Yaskawa INFORM job: OK_R2_O50&56(110_90,0)AWOK.JBI

/JOB
//NAME OK_R2_O50&56(110_90,0)AWOK
///FOLDERNAME X4
//POS
///NPOS 283,283,283,16,0,0
///TOOL 0
///POSTYPE PULSE
///PULSE
C00000=-174960,-106597,-120103,-3797,95090,7084
C00001=-145942,12948,-48978,-9200,114636,15117
C00002=-148771,199,-24149,-7829,92768,15748
C00003=-149791,3169,-18240,-7666,90580,15544
C00004=-150189,4428,-15804,-7606,89698,15465
C00005=-150189,4377,-14625,-7604,88953,15510
C00006=-150189,4428,-15804,-7606,89698,15465
C00007=-147129,1088,-19588,-8038,90597,16430
C00008=-146286,3274,-14174,-8147,88492,16849
C00009=-147032,3892,-13646,-8045,88411,16604
C00010=-146286,3274,-14174,-8147,88492,16849
C00011=-145329,9981,-8228,-8277,88377,17179
C00012=-145001,12478,-5992,-8324,88322,17293
C00013=-145329,9981,-8228,-8277,88377,17179
C00014=-145885,10408,-7967,-8202,88379,16992
C00015=-146004,9179,-11468,-8189,89874,16853
C00016=-148771,199,-24149,-7829,92768,15748
C00017=-146250,12959,-11588,-41426,106240,56782
C00018=-148467,10115,-11951,-41164,104276,56589
C00019=-154824,5653,-21154,-31285,103371,55685
C00020=-154824,5441,-20026,-31169,102684,55881
C00021=-149371,9046,-12025,-41064,103475,56508
C00022=-146311,6118,-11326,-40674,103401,57916
C00023=-147454,7095,-10477,-40693,102859,57619
C00024=-146311,6118,-11326,-40674,103401,57916
C00025=-146151,4867,-13193,-40766,103863,57802
C00026=-146384,3242,-14587,-40774,103772,57733
C00027=-146151,4867,-13193,-40766,103863,57802
C00028=-145246,5991,-13096,-40848,104676,57882
C00029=-143030,9240,-15326,-41491,108018,57509
C00030=-124603,-47737,-34158,19131,104982,-62056
C00031=-121442,-51513,-32422,19687,101389,-61480
C00032=-118855,-51471,-32397,20347,100766,-60636
C00033=-118855,-50574,-30118,20274,99880,-60787
C00034=-118855,-51471,-32397,20347,100766,-60636
C00035=-121442,-51513,-32422,19687,101389,-61480
C00036=-121797,-50324,-29168,19487,100158,-61813
C00037=-120620,-50331,-29171,19792,99877,-61431
C00038=-121797,-50324,-29168,19487,100158,-61813
C00039=-121442,-51513,-32422,19687,101389,-61480
C00040=-121603,-51176,-29855,19536,100099,-61752
C00041=-121615,-53238,-31000,19508,99766,-61811
C00042=-121603,-51176,-29855,19536,100099,-61752
C00043=-122128,-47866,-34232,19785,104374,-61232
C00044=-84141,-29178,-36607,14646,114104,-67707
C00045=-82791,-33286,-36430,14724,111710,-67503
C00046=-82229,-34853,-36282,14765,110740,-67415
C00047=-82178,-34515,-34630,14688,109914,-67503
C00048=-82229,-34853,-36282,14765,110740,-67415
C00049=-79147,-30434,-31070,15425,109262,-66446
C00050=-78452,-32631,-32544,15567,108914,-66232
C00051=-79147,-30434,-31070,15425,109262,-66446
C00052=-79730,-28966,-31252,15378,110209,-66539
C00053=-81132,-25108,-31519,15285,112547,-66756
C00054=-131359,-62866,-74976,11014,90207,-78232
C00055=-138536,21396,-13882,13391,108121,-66751
C00056=-115516,26685,-4177,3986,97138,-31002
C00057=-94522,36317,14190,8701,90062,-23707
C00058=-87387,60420,45294,7806,89491,-21265
C00059=-87081,59268,47156,7800,87741,-21270
C00060=-87136,59191,47136,7801,87720,-21290
C00061=-87136,59626,48812,7802,86921,-21339
C00062=-87136,58571,44510,7803,89008,-21209
C00063=-94386,48885,37947,21340,84274,-24043
C00064=-93739,49715,38851,21295,83986,-23861
C00065=-94392,49010,38218,21343,84180,-24062
C00066=-94392,48026,33496,21296,86424,-23665
C00067=-99028,41403,18475,21708,93080,-24149
C00068=-102045,-22247,-40217,22084,97043,-24505
C00069=-74840,-13391,-38223,2617,97503,-17820
C00070=-66507,5010,-12577,-6934,97902,-16018
C00071=-66195,5774,-8292,-6895,95700,-15788
C00072=-66101,6043,-7102,-6886,95120,-15724
C00073=-66101,6129,-6115,-6879,94563,-15693
C00074=-66101,5877,-9999,-6916,96808,-15817
C00075=-80836,-17286,-23478,14204,80508,-20001
C00076=-80064,-16344,-22775,14064,80424,-19740
C00077=-80850,-17465,-25526,14169,81645,-19874
C00078=-68799,5840,-15749,-112,106098,-15895
C00079=-55050,-26211,-40797,896,104976,-11120
C00080=-53240,-26394,-33808,1003,100562,-10527
C00081=-53174,-26119,-32540,1008,99922,-10509
C00082=-53174,-26003,-31510,1007,99347,-10512
C00083=-53450,-26813,-34326,989,100667,-10598
C00084=-66076,-50527,-45741,15470,82986,-15464
C00085=-65365,-49438,-45112,15396,83017,-15209
C00086=-66444,-51488,-48366,15481,84138,-15447
C00087=-76298,-64666,-67677,16335,90985,-18012
C00088=-121005,-146046,-93198,13283,20086,50099
C00089=-121076,-175637,-121627,12100,22333,50657
C00090=-121076,-175637,-121627,12100,22333,50657
C00091=-119842,-145846,-119955,-19490,98596,-44269
C00092=-120072,-86643,-91493,-20899,110694,-78316
C00093=-121200,-92303,-90459,-20559,107088,-78084
C00094=-138616,-107413,-91097,-21806,95703,-82500
C00095=-138616,-107085,-90210,-21788,95350,-82435
C00096=-138616,-107413,-91097,-21806,95703,-82500
C00097=-139134,-110877,-92284,-21800,94587,-82488
C00098=-138616,-107413,-91097,-21806,95703,-82500
C00099=-138504,-107678,-93902,-21887,97214,-82736
C00100=-111033,-68243,-79959,-15660,119373,-68405
C00101=-111039,-68171,-79817,-15653,119324,-68399
C00102=-111039,-68347,-78629,-15518,118531,-68280
C00103=-111039,-68171,-79817,-15653,119324,-68399
C00104=-110811,-71611,-81502,-15474,118663,-68211
C00105=-111039,-68171,-79817,-15653,119324,-68399
C00106=-117681,-73428,-89845,-994,113898,-68956
C00107=-117328,-75555,-88746,-937,112132,-68814
C00108=-117314,-76363,-88422,-931,111517,-68804
C00109=-117314,-76477,-87912,-929,111141,-68802
C00110=-117314,-76038,-89659,-939,112445,-68812
C00111=-117225,-80228,-90181,-914,110615,-68766
C00112=-117357,-73687,-89896,-955,113798,-68838
C00113=-117304,-75426,-92745,-956,114658,-68828
C00114=-117163,-75550,-92733,-938,114587,-68776
C00115=-117163,-75975,-91679,-932,113721,-68770
C00116=-117163,-75740,-92281,-935,114212,-68773
C00117=-117065,-80067,-94252,-916,113200,-68731
C00118=-117163,-75740,-92281,-935,114212,-68773
C00119=-126928,-93462,-104099,21125,97375,-56056
C00120=-123436,-95743,-101732,20630,94052,-55403
C00121=-119720,-93386,-98939,20195,92672,-54328
C00122=-119720,-93542,-97538,20172,91785,-54475
C00123=-119720,-93459,-98367,20185,92306,-54389
C00124=-117930,-93370,-98332,19971,91899,-53827
C00125=-119720,-93459,-98367,20185,92306,-54389
C00126=-119671,-100746,-101187,20141,90406,-54690
C00127=-119720,-93459,-98367,20185,92306,-54389
C00128=-121215,-96042,-102269,20389,93677,-54685
C00129=-124737,-93931,-104706,20902,96960,-55358
C00130=-120615,-97600,-94225,24394,68229,-41312
C00131=-121614,-94302,-98325,24715,72989,-35072
C00132=-121413,-94319,-98186,24655,72844,-35027
C00133=-121413,-94400,-96939,24754,72105,-35186
C00134=-121413,-94319,-98186,24655,72844,-35027
C00135=-119573,-94306,-98179,23998,72315,-34443
C00136=-121413,-94319,-98186,24655,72844,-35027
C00137=-131582,-92162,-101045,27739,78553,-37534
C00138=-149979,-79190,-101251,32758,90741,-41130
C00139=-131734,108486,68329,27886,77598,-37823
C00140=-131746,115175,77213,28093,75801,-38268
C00141=-128705,103754,56939,17355,80936,-37498
C00142=-126391,103513,58781,16629,79272,-36943
C00143=-126391,103204,59430,16657,78740,-37018
C00144=-126391,103325,59164,16645,78953,-36987
C00145=-131461,101888,64135,32515,75623,-37675
C00146=-130460,102804,65331,32242,75027,-37451
C00147=-132956,104856,68008,33106,75465,-38321
C00148=-123747,88520,39161,14959,81804,-36039
C00149=-123722,90598,43933,15013,79993,-36251
C00150=-123722,90479,44118,15020,79823,-36272
C00151=-123708,91557,46446,15056,78971,-36374
C00152=-123735,88704,42579,15029,79860,-36272
C00153=-122122,90222,44481,14459,79203,-35813
C00154=-121873,91643,46282,14382,78796,-35780
C00155=-122407,90627,44476,14554,79458,-35880
C00156=-127598,110669,63569,17480,87727,-36370
C00157=-127458,127775,88290,17571,81562,-37206
C00158=-126717,107110,60862,17217,87970,-36047
C00159=-121872,67125,15966,8400,79107,-26604
C00160=-119947,67886,17918,7577,78131,-26061
C00161=-121414,74104,25465,6223,76455,-25162
C00162=-123564,69808,18958,7132,78404,-25740
C00163=-121169,67878,17908,8113,78241,-26441
C00164=-119911,67888,17920,7562,78127,-26050
C00165=-118039,62377,14643,6757,77165,-25512
C00166=-118781,60315,11658,7068,77995,-25701
C00167=-123961,59152,819,9198,84481,-26863
C00168=-132618,-110497,-108947,28734,74981,-37704
C00169=-124566,-101520,-102656,26093,73034,-35072
C00170=-120616,-96463,-99082,24682,72208,-33752
C00171=-122368,-97019,-90544,25347,66960,-42290
C00172=-120612,-98338,-92224,24658,66756,-41637
C00173=-120867,-94497,-89822,24667,67282,-41619
C00174=-120867,-94581,-89855,24671,67261,-41624
C00175=-125926,-44970,-69160,31039,100350,-58621
C00176=-113068,-21348,-59770,17386,114865,-66123
C00177=-116612,-26527,-62656,17238,114697,-67420
C00178=-116612,-22676,-66743,18014,118989,-66712
C00179=-96791,-67830,-88966,12124,96584,-58954
C00180=-96132,-69249,-87303,11968,94777,-58911
C00181=-126837,-94677,-94277,15990,96379,-69031
C00182=-126113,-98665,-96629,15951,95659,-68871
C00183=-122876,-86143,-90735,14433,101585,-73815
C00184=-123356,-88352,-92131,14143,100582,-73012
C00185=-123771,-89216,-91995,14110,100142,-73211
C00186=-120613,-99078,-98492,7508,100072,-69302
C00187=-121484,-95136,-96163,7500,100739,-69561
C00188=-172923,-99461,-89995,9994,101945,-90389
C00189=-177663,-102072,-90824,8800,99779,-89697
C00190=-154720,-73630,-87216,6031,109011,-80641
C00191=-161015,-76454,-86164,5490,107360,-82931
C00192=-120149,-70168,-111353,-20212,74375,-72326
C00193=-120057,-133921,-120473,-34069,36215,-62022
C00194=-120146,-106815,-117651,-27009,46787,-66237
C00195=-120793,-117832,-87628,-5856,54262,2374
C00196=-128370,-47930,-37102,-5352,91873,78331
C00197=-120655,-51136,-30966,-4745,86952,81146
C00198=-120656,-51126,-30961,-4745,86954,81145
C00199=-121240,-72948,-42427,-4950,70443,81585
C00200=-120654,-52833,-32998,-4744,87329,81132
C00201=-120662,-49043,-29779,-4745,87295,81131
C00202=-130317,-72190,-42085,-4090,70120,78412
C00203=-120656,-51164,-30982,-4745,86947,81145
C00204=-120655,-51174,-30987,-4745,86946,81146
C00205=-120663,-45936,-34749,-4755,91934,80956
C00206=-120658,-53922,-38518,13016,106165,-78731
C00207=-120658,-51068,-30928,12795,103038,-79070
C00208=-120848,-68568,-43477,12343,92645,-80201
C00209=-120664,-48985,-29748,12815,103375,-79036
C00210=-120728,-51718,-32595,12818,103725,-79022
C00211=-121033,-67565,-42727,12320,93337,-80192
C00212=-120658,-51052,-30919,12796,103041,-79070
C00213=-120658,-51066,-30927,12796,103039,-79070
C00214=-93952,-51121,-30967,10241,104523,67822
C00215=-93953,-51118,-30965,10240,104524,67822
C00216=-94232,-51834,-31148,10139,104305,67705
C00217=-94418,-49164,-29853,10109,104897,67688
C00218=-92862,-50813,-31445,10614,104829,68238
C00219=-94060,-51719,-30968,10193,104235,67762
C00220=-94696,-51466,-31161,9999,104558,67560
C00221=-98759,-53921,-36367,8775,106946,66293
C00222=-98759,-54646,-38349,8822,107784,66355
C00223=-121493,-81341,-55216,13751,94719,-44592
C00224=-114524,-75581,-43376,14967,89304,-42820
C00225=-114061,-74120,-39769,15046,87799,-42845
C00226=-113295,-83137,-43502,15198,85402,-42879
C00227=-116252,-82247,-47187,14646,88567,-43499
C00228=-99157,-63031,-38155,9295,97620,-77423
C00229=-98614,-64282,-34857,9364,94917,-77440
C00230=-110866,-75942,-40129,15794,87673,-68088
C00231=-113165,-74166,-45037,15395,91900,-68341
C00232=-115008,-93546,-53723,13756,68589,-42068
C00233=-109675,-90309,-49025,11903,66648,-40175
C00234=-110872,-80814,-45342,11782,69375,-40325
C00235=-112821,-83961,-50903,11792,71421,-40812
C00236=-114232,-64224,-42018,11630,76204,-40845
C00237=-112624,-62061,-36751,11627,73886,-40501
C00238=-113161,-53891,-32402,11587,75454,-40540
C00239=-113879,-55267,-35641,11577,76817,-40664
C00240=-113966,-53043,-33005,11293,67484,-41540
C00241=-113291,-51178,-29635,11252,66296,-41408
C00242=-111200,-67941,-30076,11904,38840,-43371
C00243=-111272,-77572,-36344,12238,37781,-43569
C00244=-113557,-84331,-43308,13484,38921,-44582
C00245=-133973,-53757,-47716,12346,87026,-46675
C00246=-129752,5359,-5798,12169,90869,-44838
C00247=-101428,28800,15882,9988,85688,-35567
C00248=-103132,47107,43189,16119,89135,-35884
C00249=-99450,49923,51004,13643,85811,-34910
C00250=-98318,51183,54832,12467,84276,-34612
C00251=-99288,68654,77996,15757,90520,-34517
C00252=-98992,74868,80904,12799,90779,-34103
C00253=-96791,41543,38982,5928,76991,-34003
C00254=-97878,44550,47507,8946,72643,-34750
C00255=-97185,38348,42912,6234,63200,-34944
C00256=-98517,44066,39434,8945,77716,-34604
C00257=-111144,20698,6526,10204,87348,-38221
C00258=-130084,-64485,-54304,-2273,113857,54958
C00259=-135702,-112222,-73528,-4007,100958,53286
C00260=-120769,-181151,-111215,14764,18314,76550
C00261=-120640,-138568,-90587,5858,51266,81202
C00262=-123296,-138495,-91633,6738,52143,80161
C00263=-123889,-136810,-89749,6972,51900,79897
C00264=-120633,-141342,-91187,5942,50214,81142
C00265=-120643,-139926,-92272,5831,51603,81221
C00266=-121745,-137070,-89701,6235,51567,80759
C00267=-120643,-138359,-90541,5852,51344,81205
C00268=-120570,-183210,-103452,7665,36335,80095
C00269=-119308,-165881,-106719,1996,57355,72009
C00270=-109869,-45866,-56966,-18045,115487,59616
C00271=-130987,-55584,-53237,-19290,105982,56817
C00272=-130524,-55332,-52815,-19190,105967,56994
C00273=-130915,-50125,-47347,-17112,107567,60548
C00274=-130604,-47682,-48657,-17280,109605,60359
C00275=-169258,-4893,-18777,-15689,114847,72648
C00276=-166801,-18983,-28158,-19133,106397,68404
C00277=-169222,-12839,-23543,-16412,110304,74041
C00278=-170513,-11040,-22155,-13709,112703,78515
C00279=-163152,-15494,-28673,-22809,109474,81034
C00280=-145808,-32561,-45757,-19960,115563,86659
C00281=-146496,-66488,-70797,-11792,97357,89419
C00282=643,-91494,-100294,9175,50730,-69485
BC00000=361166,761929,143957
BC00001=361166,786367,39260
BC00002=282539,833450,219402
BC00003=282539,833450,219402
BC00004=282539,833450,219402
BC00005=282539,833450,219402
BC00006=282539,833450,219402
BC00007=282539,833450,219402
BC00008=282539,833450,219402
BC00009=282539,833450,219402
BC00010=282539,833450,219402
BC00011=282539,833450,219402
BC00012=282539,833450,219402
BC00013=282539,833450,219402
BC00014=282539,833450,219402
BC00015=282539,833450,219402
BC00016=282539,833450,219402
BC00017=320549,762407,133776
BC00018=320549,762407,133776
BC00019=320549,762407,133776
BC00020=320549,762407,133776
BC00021=320549,762407,133776
BC00022=320549,762407,133776
BC00023=320549,762407,133776
BC00024=320549,762407,133776
BC00025=320549,762407,133776
BC00026=320549,762407,133776
BC00027=320549,762407,133776
BC00028=320549,762407,133776
BC00029=320549,762407,146029
BC00030=282952,818505,325901
BC00031=282952,818505,325901
BC00032=282952,818505,325901
BC00033=282952,818505,325901
BC00034=282952,818505,325901
BC00035=282952,818505,325901
BC00036=282952,818505,325901
BC00037=282952,818505,325901
BC00038=282952,818505,325901
BC00039=282952,818505,325901
BC00040=282952,818505,325901
BC00041=282952,818505,325901
BC00042=282952,818505,325901
BC00043=282952,818505,325901
BC00044=306645,821435,249923
BC00045=306645,821435,249923
BC00046=306645,821435,249923
BC00047=306645,821435,249923
BC00048=306645,821435,249923
BC00049=306645,821435,249923
BC00050=306645,821435,249923
BC00051=306645,821435,249923
BC00052=306645,821435,249923
BC00053=306645,821435,249923
BC00054=315475,825146,222717
BC00055=328966,830815,181153
BC00056=337527,814962,251141
BC00057=285451,814962,251141
BC00058=266349,814962,251141
BC00059=266349,814962,251141
BC00060=266349,814962,251141
BC00061=266349,814962,251141
BC00062=266349,814962,251141
BC00063=266349,814962,251141
BC00064=266349,814962,251141
BC00065=266349,814962,251141
BC00066=266349,814962,251141
BC00067=266349,814962,251141
BC00068=266349,814962,251141
BC00069=266349,814962,251141
BC00070=266349,814962,251141
BC00071=266349,814962,251141
BC00072=266349,814962,251141
BC00073=266349,814962,251141
BC00074=266349,814962,251141
BC00075=266349,814962,251141
BC00076=266349,814962,251141
BC00077=266349,814962,251141
BC00078=266349,814962,251141
BC00079=266349,814962,251141
BC00080=266349,814962,251141
BC00081=266349,814962,251141
BC00082=266349,814962,251141
BC00083=266349,814962,251141
BC00084=266349,814962,251141
BC00085=266349,814962,251141
BC00086=266349,814962,251141
BC00087=266349,814962,251141
BC00088=337527,696129,251141
BC00089=337527,696129,1074810
BC00090=337527,696129,1074810
BC00091=22806,847075,1075175
BC00092=22806,847075,1075175
BC00093=22806,847075,1075175
BC00094=22806,847075,1075174
BC00095=22806,847075,1075174
BC00096=22806,847075,1075174
BC00097=22806,847075,1075174
BC00098=22806,847075,1075174
BC00099=22806,847075,1075174
BC00100=22806,847075,1075175
BC00101=22806,847075,1075175
BC00102=22806,847075,1075175
BC00103=22806,847075,1075175
BC00104=22806,847075,1075175
BC00105=22806,847075,1075175
BC00106=22806,847075,1075175
BC00107=22806,847075,1075175
BC00108=22806,847075,1075175
BC00109=22806,847075,1075175
BC00110=22806,847075,1075175
BC00111=22806,847075,1075175
BC00112=22806,847075,1075175
BC00113=60920,867427,1075175
BC00114=60920,867427,1075175
BC00115=60920,867427,1075175
BC00116=60920,867427,1075175
BC00117=60920,867427,1075175
BC00118=60920,867427,1075175
BC00119=33831,857387,1075175
BC00120=33831,857387,1075175
BC00121=33831,857387,1075175
BC00122=33831,857387,1075175
BC00123=33831,857387,1075175
BC00124=33831,857387,1075175
BC00125=33831,857387,1075175
BC00126=33831,857387,1075175
BC00127=33831,857387,1075175
BC00128=33831,857387,1075175
BC00129=33831,857387,1075175
BC00130=24152,813264,1075175
BC00131=29575,856859,1075175
BC00132=29575,856859,1075175
BC00133=29575,856859,1075175
BC00134=29575,856859,1075175
BC00135=29575,856859,1075175
BC00136=29575,856859,1075175
BC00137=29575,856859,1075175
BC00138=29575,856859,1075175
BC00139=29575,673600,1075175
BC00140=47593,737391,1075172
BC00141=47593,747171,1075172
BC00142=47593,747171,1075172
BC00143=47593,747171,1075172
BC00144=47593,747171,1075172
BC00145=47593,747171,1075172
BC00146=47593,747172,1075169
BC00147=47593,747172,1075169
BC00148=47593,747172,1075169
BC00149=47593,747172,1075166
BC00150=47593,747172,1075166
BC00151=47593,747172,1075166
BC00152=47593,747172,1075166
BC00153=47593,747172,1075166
BC00154=47593,747172,1075166
BC00155=47593,747172,1075166
BC00156=47593,747172,1075163
BC00157=47593,747172,1075163
BC00158=47593,759822,1075163
BC00159=47593,759822,1075163
BC00160=47593,759822,1075163
BC00161=47593,759822,1075159
BC00162=47593,759822,1075159
BC00163=47593,759822,1075163
BC00164=47593,759822,1075163
BC00165=47593,759822,1075163
BC00166=47593,759822,1075163
BC00167=47593,759823,1075160
BC00168=30665,865624,1075175
BC00169=30665,865624,1075175
BC00170=30665,865624,1075175
BC00171=31902,817615,1075175
BC00172=31902,817615,1075175
BC00173=31866,819043,1075175
BC00174=31866,819043,1075175
BC00175=31866,819043,1075175
BC00176=31866,819043,1075175
BC00177=31866,819043,1075175
BC00178=31866,819043,1075175
BC00179=15,838768,1075175
BC00180=15,838768,1075175
BC00181=15,836828,1075175
BC00182=15,836828,1075175
BC00183=15,838768,1075171
BC00184=790,839372,1075171
BC00185=790,839372,1075171
BC00186=7910,845642,1075175
BC00187=7910,845642,1075175
BC00188=790,839372,1075171
BC00189=790,839372,1075171
BC00190=15,812230,1075175
BC00191=15,815082,1075175
BC00192=22806,745507,951681
BC00193=22806,690051,951681
BC00194=22806,673624,951681
BC00195=349265,726928,347160
BC00196=350026,798312,408510
BC00197=350026,798312,408510
BC00198=349339,794712,384875
BC00199=349065,793272,375422
BC00200=349065,793272,375422
BC00201=349065,793272,375422
BC00202=349065,793272,375422
BC00203=336056,794671,384901
BC00204=336742,798271,408535
BC00205=336742,798271,408535
BC00206=360208,830252,356787
BC00207=361892,824921,338291
BC00208=362566,822788,330892
BC00209=362566,822788,330892
BC00210=362566,822788,330892
BC00211=368343,822804,331885
BC00212=367669,824938,339286
BC00213=365985,830270,357783
BC00214=354060,840542,361277
BC00215=351850,835820,341430
BC00216=350966,833931,333491
BC00217=350966,833931,333491
BC00218=350966,833931,333491
BC00219=354485,833948,312858
BC00220=355396,835837,320637
BC00221=357605,840559,340484
BC00222=357605,840559,340484
BC00223=357605,840559,340484
BC00224=357605,840559,340484
BC00225=357605,840559,340484
BC00226=357605,840559,340484
BC00227=357605,840559,340484
BC00228=357605,840559,340484
BC00229=357605,840559,340484
BC00230=357605,840559,340484
BC00231=357605,840559,340484
BC00232=357605,840559,340483
BC00233=357605,840559,340483
BC00234=357605,840559,340483
BC00235=357605,840559,340483
BC00236=357605,840559,340483
BC00237=357605,840559,340483
BC00238=357605,840559,340483
BC00239=357605,840559,340483
BC00240=357605,840559,340483
BC00241=357605,840559,340483
BC00242=357605,840559,340483
BC00243=357605,840559,340483
BC00244=357605,840559,340483
BC00245=357605,840559,340483
BC00246=357605,840559,340483
BC00247=301980,821787,340483
BC00248=301980,821787,340483
BC00249=301980,821788,340482
BC00250=301980,821788,340482
BC00251=301980,821788,340482
BC00252=301980,821788,340482
BC00253=301980,821788,340482
BC00254=301980,821788,340482
BC00255=301980,821788,340482
BC00256=301980,821788,340482
BC00257=301980,821788,340482
BC00258=354060,840542,361277
BC00259=354060,780758,361277
BC00260=124914,749697,239660
BC00261=124914,807441,239660
BC00262=125879,807455,202164
BC00263=125879,807455,202164
BC00264=125879,807455,202164
BC00265=125879,807455,202164
BC00266=175426,807607,202070
BC00267=175150,807603,212783
BC00268=175150,807603,212783
BC00269=238371,807603,212783
BC00270=238371,807603,212783
BC00271=238371,807603,212783
BC00272=238371,807603,212783
BC00273=238371,807603,212783
BC00274=238371,807603,212783
BC00275=303958,807603,212783
BC00276=303958,807603,212783
BC00277=303958,807603,212783
BC00278=303958,807603,212783
BC00279=303958,807603,212783
BC00280=303958,807603,212783
BC00281=311589,725441,269963
BC00282=157461,666702,53
EC00000=798156,0
EC00001=798156,0
EC00002=798156,0
EC00003=798156,0
EC00004=798156,0
EC00005=798156,0
EC00006=798156,0
EC00007=798156,0
EC00008=798156,0
EC00009=798156,0
EC00010=798156,0
EC00011=798156,0
EC00012=798156,0
EC00013=798156,0
EC00014=798156,0
EC00015=798156,0
EC00016=798156,0
EC00017=798156,0
EC00018=798156,0
EC00019=798156,0
EC00020=798156,0
EC00021=798156,0
EC00022=798156,0
EC00023=798156,0
EC00024=798156,0
EC00025=798156,0
EC00026=798156,0
EC00027=798156,0
EC00028=798156,0
EC00029=798156,0
EC00030=798156,0
EC00031=798156,0
EC00032=798156,0
EC00033=798156,0
EC00034=798156,0
EC00035=798156,0
EC00036=798156,0
EC00037=798156,0
EC00038=798156,0
EC00039=798156,0
EC00040=798156,0
EC00041=798156,0
EC00042=798156,0
EC00043=798156,0
EC00044=798156,0
EC00045=798156,0
EC00046=798156,0
EC00047=798156,0
EC00048=798156,0
EC00049=798156,0
EC00050=798156,0
EC00051=798156,0
EC00052=798156,0
EC00053=798156,0
EC00054=798156,0
EC00055=798156,0
EC00056=798156,0
EC00057=798156,0
EC00058=798156,0
EC00059=798156,0
EC00060=798156,0
EC00061=798156,0
EC00062=798156,0
EC00063=798156,0
EC00064=798156,0
EC00065=798156,0
EC00066=798156,0
EC00067=798156,0
EC00068=798156,0
EC00069=798156,0
EC00070=798156,0
EC00071=798156,0
EC00072=798156,0
EC00073=798156,0
EC00074=798156,0
EC00075=798156,0
EC00076=798156,0
EC00077=798156,0
EC00078=798156,0
EC00079=798156,0
EC00080=798156,0
EC00081=798156,0
EC00082=798156,0
EC00083=798156,0
EC00084=798156,0
EC00085=798156,0
EC00086=798156,0
EC00087=798156,0
EC00088=798156,0
EC00089=798156,0
EC00090=975524,0
EC00091=975524,0
EC00092=975524,0
EC00093=975524,0
EC00094=975522,1
EC00095=975522,1
EC00096=975522,1
EC00097=975522,1
EC00098=975522,1
EC00099=975522,1
EC00100=975524,0
EC00101=975524,0
EC00102=975524,0
EC00103=975524,0
EC00104=975524,0
EC00105=975524,0
EC00106=975524,0
EC00107=975524,0
EC00108=975524,0
EC00109=975524,0
EC00110=975524,0
EC00111=975524,0
EC00112=975524,0
EC00113=975524,0
EC00114=975524,0
EC00115=975524,0
EC00116=975524,0
EC00117=975524,0
EC00118=975524,0
EC00119=975524,0
EC00120=975524,0
EC00121=975524,0
EC00122=975524,0
EC00123=975524,0
EC00124=975524,0
EC00125=975524,0
EC00126=975524,0
EC00127=975524,0
EC00128=975524,0
EC00129=975524,0
EC00130=975524,0
EC00131=975524,0
EC00132=975524,0
EC00133=975524,0
EC00134=975524,0
EC00135=975524,0
EC00136=975524,0
EC00137=975524,0
EC00138=798157,0
EC00139=798157,0
EC00140=798155,1
EC00141=798155,1
EC00142=798155,1
EC00143=798155,1
EC00144=798155,1
EC00145=798155,1
EC00146=798154,1
EC00147=798154,1
EC00148=798154,1
EC00149=798153,1
EC00150=798153,1
EC00151=798153,1
EC00152=798153,1
EC00153=798153,1
EC00154=798153,1
EC00155=798153,1
EC00156=798152,2
EC00157=798152,2
EC00158=798152,2
EC00159=798152,2
EC00160=798152,2
EC00161=798151,2
EC00162=798151,2
EC00163=798152,2
EC00164=798152,2
EC00165=798152,2
EC00166=798152,2
EC00167=798151,2
EC00168=975524,0
EC00169=975524,0
EC00170=975524,0
EC00171=975524,0
EC00172=975524,0
EC00173=975524,0
EC00174=975524,0
EC00175=975524,0
EC00176=975524,0
EC00177=975524,0
EC00178=975524,0
EC00179=975524,0
EC00180=975524,0
EC00181=975524,0
EC00182=975524,0
EC00183=975521,1
EC00184=975521,1
EC00185=975521,1
EC00186=975524,0
EC00187=975524,0
EC00188=975521,1
EC00189=975521,1
EC00190=975524,0
EC00191=975524,0
EC00192=975524,0
EC00193=975524,0
EC00194=798156,0
EC00195=798156,0
EC00196=798156,0
EC00197=798156,0
EC00198=798156,0
EC00199=798156,0
EC00200=798156,0
EC00201=798156,0
EC00202=798156,0
EC00203=798156,0
EC00204=798156,0
EC00205=798156,0
EC00206=798156,0
EC00207=798156,0
EC00208=798156,0
EC00209=798156,0
EC00210=798156,0
EC00211=798154,1
EC00212=798156,0
EC00213=798156,0
EC00214=798156,0
EC00215=798156,0
EC00216=798156,0
EC00217=798156,0
EC00218=798156,0
EC00219=798156,0
EC00220=798156,0
EC00221=798156,0
EC00222=798156,0
EC00223=798156,0
EC00224=798156,0
EC00225=798156,0
EC00226=798156,0
EC00227=798156,0
EC00228=798156,0
EC00229=798156,0
EC00230=798156,0
EC00231=798156,0
EC00232=798155,0
EC00233=798155,0
EC00234=798155,0
EC00235=798155,0
EC00236=798155,0
EC00237=798155,0
EC00238=798155,0
EC00239=798155,0
EC00240=798155,0
EC00241=798155,0
EC00242=798155,0
EC00243=798155,0
EC00244=798155,0
EC00245=798155,0
EC00246=798155,0
EC00247=798155,0
EC00248=798155,0
EC00249=798154,0
EC00250=798154,0
EC00251=798154,0
EC00252=798154,0
EC00253=798154,0
EC00254=798154,0
EC00255=798154,0
EC00256=798154,0
EC00257=798154,0
EC00258=798156,0
EC00259=798156,0
EC00260=798156,0
EC00261=798156,0
EC00262=798156,0
EC00263=798156,0
EC00264=798156,0
EC00265=798156,0
EC00266=798156,0
EC00267=798156,0
EC00268=798156,0
EC00269=798156,0
EC00270=798156,0
EC00271=798156,0
EC00272=798156,0
EC00273=798156,0
EC00274=798156,0
EC00275=798156,0
EC00276=798156,0
EC00277=798156,0
EC00278=798156,0
EC00279=798156,0
EC00280=798156,0
EC00281=798156,0
EC00282=798156,0
///POSTYPE BASE
///RECTAN
///RCONF 0,0,0,0,0,0,0,0,0,0,0,0,0,0,0,0,0,0,0,0,0,0,0,0
P00006=0.222,-3.123,-1.508,0.0000,0.0000,0.0000
P00023=0.143,-0.036,0.682,0.0000,0.0000,0.0000
P00024=0.145,-0.552,1.326,0.0000,0.0000,0.0000
P00025=-2.003,0.006,0.728,0.0000,0.0000,0.0000
P00026=0.562,-0.002,-0.337,0.0000,0.0000,0.0000
P00031=1.853,-0.001,-1.549,0.0000,0.0000,0.0000
P00032=1.957,0.503,-7.217,0.0000,0.0000,0.0000
///RCONF 0,0,0,0,1,0,0,0,0,0,0,0,0,0,0,0,0,0,0,0,0,0,0,0
P00033=-0.123,0.612,-5.012,0.0000,0.0000,0.0000
///RCONF 0,0,0,0,0,0,0,0,0,0,0,0,0,0,0,0,0,0,0,0,0,0,0,0
P00034=-0.304,0.773,-2.693,0.0000,0.0000,0.0000
P00040=-0.030,9.648,2.467,0.0000,0.0000,0.0000
P00044=0.687,-2.322,1.156,0.0000,0.0000,0.0000
P00050=4.296,-4.501,-0.826,0.0000,0.0000,0.0000
P00051=0.367,3.892,0.009,0.0000,0.0000,0.0000
P00052=0.088,2.832,-0.342,0.0000,0.0000,0.0000
P00060=2.327,-2.514,-2.692,0.0000,0.0000,0.0000
P00061=1.575,-3.405,-0.752,0.0000,0.0000,0.0000
//INST
///DATE 2025/01/29 12:24
///ATTR SC,RW
///GROUP1 RB1,BS1
///GROUP2 ST1
NOP
'OK_r2_O50&56(110_90,0)
'Down
MOVJ C00000 BC00000 VJ=100.00  +MOVJ EC00000 VJ=100.00
MOVJ C00001 BC00001 VJ=100.00  +MOVJ EC00001 VJ=100.00
'Path S1597
SFTOF3D
MOVJ C00002 BC00002 VJ=100.00  +MOVJ EC00002 VJ=100.00
MOVL C00003 BC00003 V=333.3  +MOVJ EC00003 VJ=100.00
SMOVL C00004 BC00004 V=100.0  +MOVJ EC00004
SREFP 3 C00005 BC00005  +REFP EC00005
CALL JOB:SEARCH-R1-S13D
SET P026 P006
SFTON3D P026
SMOVL C00006 BC00006 V=100.0  +MOVJ EC00006
SMOVL C00007 BC00007 V=333.3  +MOVJ EC00007
SMOVL C00008 BC00008 V=100.0  +MOVJ EC00008
SREFP 3 C00009 BC00009  +REFP EC00009
CALL JOB:SEARCH-R1-S13D
SET P026 P006
SFTON3D P026
SMOVL C00010 BC00010 V=100.0  +MOVJ EC00010
SMOVL C00011 BC00011 V=100.0  +MOVJ EC00011
SREFP 3 C00012 BC00012  +REFP EC00012
CALL JOB:SEARCH-R1-S13D
SET P026 P006
SFTON3D P026
SMOVL C00013 BC00013 V=100.0  +MOVJ EC00013
SMOVL C00014 BC00014 V=100.0  +MOVJ EC00014
SMOVL C00015 BC00015 V=100.0  +MOVJ EC00015
MOVL C00016 BC00016 V=1000.0  +MOVJ EC00016 VJ=100.00
'Path S1598
SFTOF3D
MOVJ C00017 BC00017 VJ=100.00  +MOVJ EC00017 VJ=100.00
MOVL C00018 BC00018 V=333.3  +MOVJ EC00018 VJ=100.00
SMOVL C00019 BC00019 V=100.0  +MOVJ EC00019
SREFP 3 C00020 BC00020  +REFP EC00020
CALL JOB:SEARCH-R1-S13D
SET P025 P006
SFTON3D P025
SMOVL C00021 BC00021 V=100.0  +MOVJ EC00021
SMOVL C00022 BC00022 V=100.0  +MOVJ EC00022
SREFP 3 C00023 BC00023  +REFP EC00023
CALL JOB:SEARCH-R1-S13D
SET P025 P006
SFTON3D P025
SMOVL C00024 BC00024 V=100.0  +MOVJ EC00024
SMOVL C00025 BC00025 V=100.0  +MOVJ EC00025
SREFP 3 C00026 BC00026  +REFP EC00026
CALL JOB:SEARCH-R1-S13D
SET P025 P006
SFTON3D P025
SMOVL C00027 BC00027 V=100.0  +MOVJ EC00027
MOVL C00028 BC00028 V=400.0  +MOVJ EC00028 VJ=100.00
MOVL C00029 BC00029 V=1000.0  +MOVJ EC00029 VJ=100.00
'Path S1599
SFTOF3D
MOVJ C00030 BC00030 VJ=100.00  +MOVJ EC00030 VJ=100.00
SMOVL C00031 BC00031 V=333.3  +MOVJ EC00031
SMOVL C00032 BC00032 V=100.0  +MOVJ EC00032
SREFP 3 C00033 BC00033  +REFP EC00033
CALL JOB:SEARCH-R1-S13D
SET P023 P006
SFTON3D P023
SMOVL C00034 BC00034 V=100.0  +MOVJ EC00034
SMOVL C00035 BC00035 V=166.7  +MOVJ EC00035
SMOVL C00036 BC00036 V=100.0  +MOVJ EC00036
SREFP 3 C00037 BC00037  +REFP EC00037
CALL JOB:SEARCH-R1-S13D
SET P023 P006
SFTON3D P023
SMOVL C00038 BC00038 V=100.0  +MOVJ EC00038
SMOVL C00039 BC00039 V=166.7  +MOVJ EC00039
SMOVL C00040 BC00040 V=100.0  +MOVJ EC00040
SREFP 3 C00041 BC00041  +REFP EC00041
CALL JOB:SEARCH-R1-S13D
SET P023 P006
SFTON3D P023
SMOVL C00042 BC00042 V=100.0  +MOVJ EC00042
MOVL C00043 BC00043 V=1000.0  +MOVJ EC00043 VJ=100.00
'Path S1600
SFTOF3D
MOVJ C00044 BC00044 VJ=100.00  +MOVJ EC00044 VJ=100.00
MOVL C00045 BC00045 V=400.0  +MOVJ EC00045 VJ=100.00
SMOVL C00046 BC00046 V=100.0  +MOVJ EC00046
SREFP 3 C00047 BC00047  +REFP EC00047
CALL JOB:SEARCH-R1-S13D
SET P024 P006
SFTON3D P024
SMOVL C00048 BC00048 V=100.0  +MOVJ EC00048
SMOVL C00049 BC00049 V=100.0  +MOVJ EC00049
SREFP 3 C00050 BC00050  +REFP EC00050
CALL JOB:SEARCH-R1-S13D
SET P024 P006
SFTON3D P024
SMOVL C00051 BC00051 V=100.0  +MOVJ EC00051
MOVL C00052 BC00052 V=400.0  +MOVJ EC00052 VJ=100.00
MOVL C00053 BC00053 V=1000.0  +MOVJ EC00053 VJ=100.00
MOVJ C00054 BC00054 VJ=100.00  +MOVJ EC00054 VJ=100.00
'Path S1601
SFTOF3D
MOVJ C00055 BC00055 VJ=100.00  +MOVJ EC00055 VJ=100.00
MOVJ C00056 BC00056 VJ=100.00  +MOVJ EC00056 VJ=40.00
MOVJ C00057 BC00057 VJ=100.00  +MOVJ EC00057 VJ=40.00
MOVJ C00058 BC00058 VJ=15.00  +MOVJ EC00058 VJ=40.00
MOVJ C00059 BC00059 VJ=10.00  +MOVJ EC00059 VJ=40.00
SMOVL C00060 BC00060 V=100.0  +MOVJ EC00060
SREFP 3 C00061 BC00061  +REFP EC00061
CALL JOB:SEARCH-R1-S13D
SET P050 P006
SFTON3D P050
SMOVL C00062 BC00062 V=83.3  +MOVJ EC00062
SMOVL C00063 BC00063 V=83.3  +MOVJ EC00063
SREFP 3 C00064 BC00064  +REFP EC00064
CALL JOB:SEARCH-R1-S13D
SET P050 P006
SFTON3D P050
SFTOF3D
SMOVL C00065 BC00065 V=100.0  +MOVJ EC00065
MOVJ C00066 BC00066 VJ=100.00  +MOVJ EC00066 VJ=10.00
MOVJ C00067 BC00067 VJ=100.00  +MOVJ EC00067 VJ=10.00
MOVJ C00068 BC00068 VJ=100.00  +MOVJ EC00068 VJ=50.00
MOVJ C00069 BC00069 VJ=100.00  +MOVJ EC00069 VJ=50.00
MOVJ C00070 BC00070 VJ=100.00  +MOVJ EC00070 VJ=50.00
MOVJ C00071 BC00071 VJ=10.00  +MOVJ EC00071 VJ=50.00
SMOVL C00072 BC00072 V=100.0  +MOVJ EC00072
SREFP 3 C00073 BC00073  +REFP EC00073
CALL JOB:SEARCH-R1-S13D
SET P051 P006
SFTON3D P051
SMOVL C00074 BC00074 V=83.3  +MOVJ EC00074
SMOVL C00075 BC00075 V=100.0  +MOVJ EC00075
SREFP 3 C00076 BC00076  +REFP EC00076
CALL JOB:SEARCH-R1-S13D
SET P051 P006
SFTON3D P051
SFTOF3D
SMOVL C00077 BC00077 V=133.3  +MOVJ EC00077
MOVJ C00078 BC00078 VJ=40.00  +MOVJ EC00078 VJ=40.00
MOVJ C00079 BC00079 VJ=100.00  +MOVJ EC00079 VJ=10.00
MOVJ C00080 BC00080 VJ=10.00  +MOVJ EC00080 VJ=40.00
SMOVL C00081 BC00081 V=100.0  +MOVJ EC00081
SREFP 3 C00082 BC00082  +REFP EC00082
CALL JOB:SEARCH-R1-S13D
SET P052 P006
SFTON3D P052
SMOVL C00083 BC00083 V=83.3  +MOVJ EC00083
SMOVL C00084 BC00084 V=100.0  +MOVJ EC00084
SREFP 3 C00085 BC00085  +REFP EC00085
CALL JOB:SEARCH-R1-S13D
SET P052 P006
SFTON3D P052
SFTOF3D
SMOVL C00086 BC00086 V=100.0  +MOVJ EC00086
MOVJ C00087 BC00087 VJ=100.00  +MOVJ EC00087 VJ=10.00
MOVJ C00088 BC00088 VJ=100.00  +MOVJ EC00088 VJ=100.00
MOVJ C00089 BC00089 VJ=100.00  +MOVJ EC00089 VJ=100.00
MOVJ C00090 BC00090 VJ=100.00  +MOVJ EC00090 VJ=100.00
'Up
MOVJ C00091 BC00091 VJ=100.00  +MOVJ EC00091 VJ=100.00
'Path S1129
SFTOF3D
MOVJ C00092 BC00092 VJ=100.00  +MOVJ EC00092 VJ=100.00
MOVL C00093 BC00093 V=400.0  +MOVJ EC00093 VJ=100.00
SMOVL C00094 BC00094 V=100.0  +MOVJ EC00094
SREFP 3 C00095 BC00095  +REFP EC00095
CALL JOB:SEARCH-R1-S13D
SET P033 P006
SFTON3D P033
SMOVL C00096 BC00096 V=100.0  +MOVJ EC00096
SREFP 3 C00097 BC00097  +REFP EC00097
CALL JOB:SEARCH-R1-S13D
SET P033 P006
SFTON3D P033
SMOVL C00098 BC00098 V=100.0  +MOVJ EC00098
SFTOF3D
SMOVL C00099 BC00099 V=166.7  +MOVJ EC00099
MOVL C00100 BC00100 V=400.0  +MOVJ EC00100 VJ=100.00
SMOVL C00101 BC00101 V=100.0  +MOVJ EC00101
SREFP 3 C00102 BC00102  +REFP EC00102
CALL JOB:SEARCH-R1-S13D
SET P034 P006
SFTON3D P034
SMOVL C00103 BC00103 V=100.0  +MOVJ EC00103
SREFP 3 C00104 BC00104  +REFP EC00104
CALL JOB:SEARCH-R1-S13D
SET P034 P006
SFTON3D P034
SMOVL C00105 BC00105 V=100.0  +MOVJ EC00105
SFTOF3D
MOVJ C00106 BC00106 VJ=100.00  +MOVJ EC00106 VJ=100.00
MOVL C00107 BC00107 V=400.0  +MOVJ EC00107 VJ=100.00
SMOVL C00108 BC00108 V=100.0  +MOVJ EC00108
SREFP 3 C00109 BC00109  +REFP EC00109
CALL JOB:SEARCH-R1-S13D
SET P032 P006
SFTON3D P032
SMOVL C00110 BC00110 V=100.0  +MOVJ EC00110
SREFP 3 C00111 BC00111  +REFP EC00111
CALL JOB:SEARCH-R1-S13D
SET P032 P006
SFTON3D P032
SMOVL C00112 BC00112 V=100.0  +MOVJ EC00112
SFTOF3D
MOVL C00113 BC00113 V=400.0  +MOVJ EC00113 VJ=100.00
SMOVL C00114 BC00114 V=100.0  +MOVJ EC00114
SREFP 3 C00115 BC00115  +REFP EC00115
CALL JOB:SEARCH-R1-S13D
SET P044 P006
SFTON3D P044
SMOVL C00116 BC00116 V=100.0  +MOVJ EC00116
SREFP 3 C00117 BC00117  +REFP EC00117
CALL JOB:SEARCH-R1-S13D
SET P044 P006
SFTON3D P044
SMOVL C00118 BC00118 V=100.0  +MOVJ EC00118
'Path S1118
SFTOF3D
MOVJ C00119 BC00119 VJ=100.00  +MOVJ EC00119 VJ=100.00
MOVL C00120 BC00120 V=400.0  +MOVJ EC00120 VJ=100.00
SMOVL C00121 BC00121 V=100.0  +MOVJ EC00121
SREFP 3 C00122 BC00122  +REFP EC00122
CALL JOB:SEARCH-R1-S13D
SET P031 P006
SFTON3D P031
SMOVL C00123 BC00123 V=100.0  +MOVJ EC00123
SREFP 3 C00124 BC00124  +REFP EC00124
CALL JOB:SEARCH-R1-S13D
SET P031 P006
SFTON3D P031
SMOVL C00125 BC00125 V=100.0  +MOVJ EC00125
SREFP 3 C00126 BC00126  +REFP EC00126
CALL JOB:SEARCH-R1-S13D
SET P031 P006
SFTON3D P031
SMOVL C00127 BC00127 V=100.0  +MOVJ EC00127
MOVL C00128 BC00128 V=400.0  +MOVJ EC00128 VJ=100.00
MOVL C00129 BC00129 V=1000.0  +MOVJ EC00129 VJ=100.00
'Path W344
SFTOF3D
MOVJ C00130 BC00130 VJ=100.00  +MOVJ EC00130 VJ=100.00
SMOVL C00131 BC00131 V=400.0  +MOVJ EC00131
SMOVL C00132 BC00132 V=100.0  +MOVJ EC00132
SREFP 3 C00133 BC00133  +REFP EC00133
CALL JOB:SEARCH-R1-S13D
SET P040 P006
SFTON3D P040
SMOVL C00134 BC00134 V=100.0  +MOVJ EC00134
SREFP 3 C00135 BC00135  +REFP EC00135
CALL JOB:SEARCH-R1-S13D
SET P040 P006
SFTON3D P040
SMOVL C00136 BC00136 V=166.7  +MOVJ EC00136
SFTOF3D
MOVJ C00137 BC00137 VJ=100.00  +MOVJ EC00137 VJ=100.00
MOVJ C00138 BC00138 VJ=100.00  +MOVJ EC00138 VJ=100.00
MOVL C00139 BC00139 V=666.7  +MOVJ EC00139 VJ=100.00
SMOVL C00140 BC00140 V=666.7  +MOVJ EC00140
SMOVL C00141 BC00141 V=400.0  +MOVJ EC00141
SMOVL C00142 BC00142 V=100.0  +MOVJ EC00142
SREFP 3 C00143 BC00143  +REFP EC00143
CALL JOB:SEARCH-R1-S13D
SET P060 P006
SFTON3D P060
SMOVL C00144 BC00144 V=100.0  +MOVJ EC00144
SMOVL C00145 BC00145 V=100.0  +MOVJ EC00145
SREFP 3 C00146 BC00146  +REFP EC00146
CALL JOB:SEARCH-R1-S13D
SET P060 P006
SFTON3D P060
SMOVL C00147 BC00147 V=166.7  +MOVJ EC00147
SFTOF3D
SMOVL C00148 BC00148 V=666.7  +MOVJ EC00148
SMOVL C00149 BC00149 V=400.0  +MOVJ EC00149
SMOVL C00150 BC00150 V=100.0  +MOVJ EC00150
SREFP 3 C00151 BC00151  +REFP EC00151
CALL JOB:SEARCH-R1-S13D
SET P061 P006
SFTON3D P061
SMOVL C00152 BC00152 V=100.0  +MOVJ EC00152
SMOVL C00153 BC00153 V=100.0  +MOVJ EC00153
SREFP 3 C00154 BC00154  +REFP EC00154
CALL JOB:SEARCH-R1-S13D
SET P061 P006
SFTON3D P061
SMOVL C00155 BC00155 V=166.7  +MOVJ EC00155
SFTOF3D
SMOVL C00156 BC00156 V=400.0  +MOVJ EC00156
SMOVL C00157 BC00157 V=400.0  +MOVJ EC00157
SMOVL C00158 BC00158 V=400.0  +MOVJ EC00158
SFTON3D P061
SMOVL C00159 BC00159 V=400.0  +MOVJ EC00159
SMOVL C00160 BC00160 V=166.7 PL=0  +MOVJ EC00160
MACRO1 MJ#(0) ARGF9
ARCON
SMOVL C00161 BC00161 V=10.0  +MOVJ EC00161
ARCOF
SMOVL C00162 BC00162 V=166.7  +MOVJ EC00162
SFTOF3D
SMOVL C00163 BC00163 V=166.7  +MOVJ EC00163
SFTON3D P061
SMOVL C00164 BC00164 V=166.7 PL=0  +MOVJ EC00164
ARCON
SMOVL C00165 BC00165 V=10.0  +MOVJ EC00165
ARCOF
SMOVL C00166 BC00166 V=166.7  +MOVJ EC00166
SFTOF3D
SMOVL C00167 BC00167 V=400.0  +MOVJ EC00167
SMOVL C00168 BC00168 V=1000.0  +MOVJ EC00168
SMOVL C00169 BC00169 V=400.0  +MOVJ EC00169
SMOVL C00170 BC00170 V=166.7 PL=0  +MOVJ EC00170
SREFP 1 C00171 BC00171  +REFP EC00171
SREFP 2 C00172 BC00172  +REFP EC00172
MACRO1 MJ#(0) ARGF9
ARCON
SFTON3D P031
SMOVL C00173 BC00173 V=8.3  +MOVJ EC00173
SMOVC C00174 BC00174 V=8.3  +MOVJ EC00174
SMOVC C00175 BC00175 V=8.3  +MOVJ EC00175
SMOVC C00176 BC00176 V=8.3  +MOVJ EC00176
SMOVL C00177 BC00177 V=8.3  +MOVJ EC00177
ARCOF
SMOVL C00178 BC00178 V=400.0  +MOVJ EC00178
SFTOF3D
SMOVL C00179 BC00179 V=400.0  +MOVJ EC00179
SFTON3D P032
SMOVL C00180 BC00180 V=133.3 PL=0  +MOVJ EC00180
SREFP 1 C00181 BC00181  +REFP EC00181
SREFP 2 C00182 BC00182  +REFP EC00182
MACRO1 MJ#(0) ARGF9
ARCON
SWVON WEV#(60)
SFTON3D P032
SMOVL C00183 BC00183 V=9.2  +MOVJ EC00183
ARCOF
SWVOF
SMOVL C00184 BC00184 V=400.0  +MOVJ EC00184
SFTOF3D
SFTON3D P034
SMOVL C00185 BC00185 V=133.3 PL=0  +MOVJ EC00185
SREFP 1 C00186 BC00186  +REFP EC00186
SREFP 2 C00187 BC00187  +REFP EC00187
MACRO1 MJ#(0) ARGF9
ARCON
SMOVL C00188 BC00188 V=9.2  +MOVJ EC00188
SMOVL C00189 BC00189 V=9.2  +MOVJ EC00189
ARCOF
SMOVL C00190 BC00190 V=400.0  +MOVJ EC00190
SMOVL C00191 BC00191 V=1000.0  +MOVJ EC00191
SFTOF3D
MOVJ C00192 BC00192 VJ=100.00  +MOVJ EC00192 VJ=100.00
MOVJ C00193 BC00193 VJ=100.00  +MOVJ EC00193 VJ=100.00
MOVJ C00194 BC00194 VJ=100.00  +MOVJ EC00194 VJ=100.00
'Down
MOVJ C00195 BC00195 VJ=100.00  +MOVJ EC00195 VJ=100.00
'Path W1603
SFTOF3D
MOVJ C00196 BC00196 VJ=100.00  +MOVJ EC00196 VJ=100.00
'Path W1605
SFTOF3D
SFTON3D P023
MOVJ C00197 BC00197 VJ=100.00  +MOVJ EC00197 VJ=100.00
SMOVL C00198 BC00198 V=1000.0  +MOVJ EC00198
SMOVL C00199 BC00199 V=133.3 PL=0  +MOVJ EC00199
SREFP 1 C00200 BC00200  +REFP EC00200
SREFP 2 C00201 BC00201  +REFP EC00201
MACRO1 MJ#(0) ARGF14
ARCON
SMOVL C00202 BC00202 V=10.8  +MOVJ EC00202
ARCOF
SMOVL C00203 BC00203 V=400.0  +MOVJ EC00203
SMOVL C00204 BC00204 V=1000.0  +MOVJ EC00204
MOVJ C00205 BC00205 VJ=100.00  +MOVJ EC00205 VJ=30.00
SFTOF3D
'Path W1606
SFTOF3D
SFTON3D P024
MOVJ C00206 BC00206 VJ=100.00  +MOVJ EC00206 VJ=100.00
SMOVL C00207 BC00207 V=1000.0  +MOVJ EC00207
SMOVL C00208 BC00208 V=133.3 PL=0  +MOVJ EC00208
SREFP 1 C00209 BC00209  +REFP EC00209
SREFP 2 C00210 BC00210  +REFP EC00210
MACRO1 MJ#(0) ARGF14
ARCON
SMOVL C00211 BC00211 V=11.7  +MOVJ EC00211
ARCOF
SMOVL C00212 BC00212 V=400.0  +MOVJ EC00212
SMOVL C00213 BC00213 V=1000.0  +MOVJ EC00213
SFTOF3D
'Path W1607
SFTOF3D
SFTON3D P024
MOVJ C00214 BC00214 VJ=100.00  +MOVJ EC00214 VJ=100.00
SMOVL C00215 BC00215 V=166.7  +MOVJ EC00215
SMOVL C00216 BC00216 V=133.3 PL=0  +MOVJ EC00216
ARCON
SREFP 1 C00217 BC00217  +REFP EC00217
SREFP 2 C00218 BC00218  +REFP EC00218
MACRO1 MJ#(0) ARGF6
SMOVL C00219 BC00219 V=13.3  +MOVJ EC00219
ARCOF
SMOVL C00220 BC00220 V=400.0  +MOVJ EC00220
SMOVL C00221 BC00221 V=1000.0  +MOVJ EC00221
MOVJ C00222 BC00222 VJ=100.00  +MOVJ EC00222 VJ=30.00
MOVJ C00223 BC00223 VJ=100.00  +MOVJ EC00223 VJ=30.00
MOVJ C00224 BC00224 VJ=30.00  +MOVJ EC00224 VJ=100.00
SFTOF3D
SFTON3D P052
MACRO1 MJ#(0) ARGF14
SMOVL C00225 BC00225 V=83.3  +MOVJ EC00225
ARCON
SMOVL C00226 BC00226 V=10.0  +MOVJ EC00226
ARCOF
SMOVL C00227 BC00227 V=166.7  +MOVJ EC00227
MOVJ C00228 BC00228 VJ=40.00  +MOVJ EC00228 VJ=70.00
SFTON3D P024
SMOVL C00229 BC00229 V=66.7  +MOVJ EC00229
ARCON
SMOVL C00230 BC00230 V=10.0  +MOVJ EC00230
ARCOF
SMOVL C00231 BC00231 V=250.0  +MOVJ EC00231
SMOVL C00232 BC00232 V=400.0  +MOVJ EC00232
SFTON3D P052
SMOVL C00233 BC00233 V=100.0  +MOVJ EC00233
ARCON
SMOVL C00234 BC00234 V=10.0  +MOVJ EC00234
ARCOF
SMOVL C00235 BC00235 V=166.7  +MOVJ EC00235
SMOVL C00236 BC00236 V=666.7  +MOVJ EC00236
SFTON3D P051
SMOVL C00237 BC00237 V=100.0  +MOVJ EC00237
ARCON
SMOVL C00238 BC00238 V=10.0  +MOVJ EC00238
ARCOF
SMOVL C00239 BC00239 V=333.3  +MOVJ EC00239
SMOVL C00240 BC00240 V=500.0  +MOVJ EC00240
SMOVL C00241 BC00241 V=100.0  +MOVJ EC00241
ARCON
SMOVL C00242 BC00242 V=10.0  +MOVJ EC00242
ARCOF
SMOVL C00243 BC00243 V=166.7  +MOVJ EC00243
SMOVL C00244 BC00244 V=1000.0  +MOVJ EC00244
SMOVL C00245 BC00245 V=1000.0  +MOVJ EC00245
SMOVL C00246 BC00246 V=1000.0  +MOVJ EC00246
SMOVL C00247 BC00247 V=1000.0  +MOVJ EC00247
SMOVL C00248 BC00248 V=400.0  +MOVJ EC00248
SMOVL C00249 BC00249 V=166.7  +MOVJ EC00249
SFTON3D P050
SMOVL C00250 BC00250 V=100.0  +MOVJ EC00250
ARCON
SMOVL C00251 BC00251 V=10.0  +MOVJ EC00251
ARCOF
SMOVL C00252 BC00252 V=133.3  +MOVJ EC00252
SMOVL C00253 BC00253 V=333.3  +MOVJ EC00253
SMOVL C00254 BC00254 V=83.3  +MOVJ EC00254
ARCON
SMOVL C00255 BC00255 V=10.0  +MOVJ EC00255
ARCOF
SMOVL C00256 BC00256 V=83.3  +MOVJ EC00256
MOVJ C00257 BC00257 VJ=100.00  +MOVJ EC00257 VJ=30.00
MOVJ C00258 BC00258 VJ=100.00  +MOVJ EC00258 VJ=100.00
MOVJ C00259 BC00259 VJ=100.00  +MOVJ EC00259 VJ=100.00
MOVJ C00260 BC00260 VJ=100.00  +MOVJ EC00260 VJ=100.00
'Path W1608
SFTOF3D
SFTON3D P025
MOVJ C00261 BC00261 VJ=100.00  +MOVJ EC00261 VJ=100.00
SMOVL C00262 BC00262 V=333.3  +MOVJ EC00262
SMOVL C00263 BC00263 V=133.3 PL=0  +MOVJ EC00263
SREFP 1 C00264 BC00264  +REFP EC00264
SREFP 2 C00265 BC00265  +REFP EC00265
MACRO1 MJ#(0) ARGF14
ARCON
SMOVL C00266 BC00266 V=11.7  +MOVJ EC00266
ARCOF
SMOVL C00267 BC00267 V=400.0  +MOVJ EC00267
SMOVL C00268 BC00268 V=1000.0  +MOVJ EC00268
SMOVL C00269 BC00269 V=1000.0  +MOVJ EC00269
SMOVL C00270 BC00270 V=1000.0  +MOVJ EC00270
SMOVL C00271 BC00271 V=166.7  +MOVJ EC00271
ARCON
SMOVL C00272 BC00272 V=12.5  +MOVJ EC00272
SMOVL C00273 BC00273 V=12.5  +MOVJ EC00273
ARCOF
SMOVL C00274 BC00274 V=133.3  +MOVJ EC00274
SMOVL C00275 BC00275 V=166.7  +MOVJ EC00275
SMOVL C00276 BC00276 V=166.7  +MOVJ EC00276
ARCON
SMOVL C00277 BC00277 V=10.8  +MOVJ EC00277
SMOVL C00278 BC00278 V=10.8  +MOVJ EC00278
ARCOF
SFTOF3D
SMOVL C00279 BC00279 V=250.0  +MOVJ EC00279
SMOVL C00280 BC00280 V=500.0  +MOVJ EC00280
MOVJ C00281 BC00281 VJ=100.00  +MOVJ EC00281 VJ=100.00
MOVJ C00282 BC00282 VJ=100.00  +MOVJ EC00282 VJ=50.00
END
